(* PLC project Unnamed, Unknown Unnamed 1 *)
(* stored: creationDateTime 2024-07-24T21:58:42, modificationDateTime 2024-07-25T08:59:15 *)

PROGRAM TrafficLights
  VAR
    Input : BOOL;
    RedN : BOOL;
    YellowN : BOOL;
    GreenN : BOOL;
    RedS : BOOL;
    YellowS : BOOL;
    GreenS : BOOL;
    M0 : BOOL;
    TP0 : TP;
    TP1 : TP;
    TP2 : TP;
    TP3 : TP;
  END_VAR

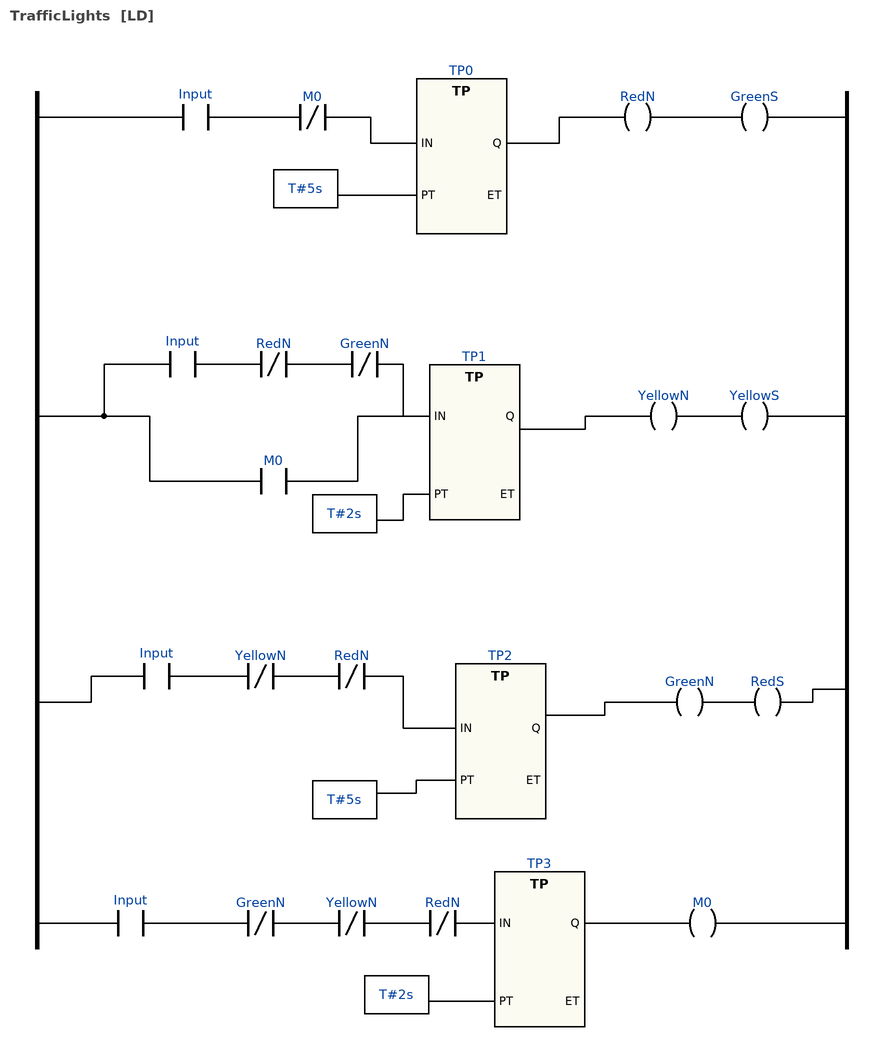
(* LD diagram, written out as Structured Text *)
TP0(IN := Input AND NOT M0, PT := T#5s);
RedN := TP0.Q;
TP1(IN := Input AND NOT RedN AND NOT GreenN OR M0, PT := T#2s);
YellowN := TP1.Q;
TP2(IN := Input AND NOT YellowN AND NOT RedN, PT := T#5s);
GreenN := TP2.Q;
TP3(IN := Input AND NOT GreenN AND NOT YellowN AND NOT RedN, PT := T#2s);
M0 := TP3.Q;
GreenS := TP0.Q;
YellowS := TP1.Q;
RedS := TP2.Q;
END_PROGRAM

CONFIGURATION Config0
  RESOURCE Res0 ON PLC
    TASK task0(INTERVAL := T#20ms, PRIORITY := 0);
    PROGRAM instance0 WITH task0 : TrafficLights;
  END_RESOURCE
END_CONFIGURATION
